INTERFACE I_Controller

METHOD Auto
VAR_INPUT
END_VAR
END_METHOD

PROPERTY Error : BOOL
GET
END_GET
SET
END_SET
END_PROPERTY

METHOD Init : BOOL
VAR_INPUT
END_VAR
END_METHOD

METHOD Manual
VAR_INPUT
END_VAR
END_METHOD

PROPERTY Mode : E_ControlMode
GET
END_GET
SET
END_SET
END_PROPERTY

METHOD Off
VAR_INPUT
END_VAR
END_METHOD

METHOD OperationTest : BOOL
VAR_INPUT
END_VAR
END_METHOD

METHOD Run
VAR_INPUT
END_VAR
END_METHOD

END_INTERFACE

(* stored: Version 1.1.0.1, ProductVersion 3.1.4024.0
   Itf I_Controller: Id {740ca180-aa21-4a42-a251-bd76d55996ea}
   Method Auto: Id {1c9ec7f1-f6d0-4d72-a520-fae895337145}
   Property Error: Id {36daf20e-43bc-4f3f-987c-778cb1b6d7bf}
   Get Get: Id {8161dd48-d5c8-4ad6-a66b-185296c23149}
   Set Set: Id {22199c3f-bac7-483c-8d6c-499588aaa150}
   Method Init: Id {826a7cdb-e9b9-4794-af63-b87a1f7833c6}
   Method Manual: Id {3aaf6c4b-9c33-407d-b7dd-757b5f27ff88}
   Property Mode: Id {f207765e-b05f-4960-a16b-3d77e49ab629}
   Get Get: Id {ffff0b8e-03ca-407d-b422-984d38e92b53}
   Set Set: Id {bc90e767-6510-4ff7-9505-75454838d4a2}
   Method Off: Id {dec2e242-dde5-41ca-a249-e829027fa7d7}
   Method OperationTest: Id {ada3f3a2-7656-4a39-b127-408ce5ba258d}
   Method Run: Id {79918f9b-ec4b-463e-9880-9502a5639904} *)
